{attribute 'linkalways'} 
{attribute 'no_explicit_call' := 'This FB is a CLASS and must be accessed using methods or properties'}
{attribute 'enable_dynamic_creation'}
FUNCTION_BLOCK _ETcVnDrawMatchesFlags EXTENDS EnumDatatypeBase
VAR
	localData : ETcVnDrawMatchesFlags;
	activeData : REFERENCE TO ETcVnDrawMatchesFlags;
	enumBaseDatatype : _DINT(localData);
END_VAR

METHOD PRIVATE AddLocalEnumeration
VAR_INPUT
	Enumeration : T_MAXSTRING;
	Value : ETcVnDrawMatchesFlags;
END_VAR
AddEnumeration(Enumeration, Value);
END_METHOD

PROPERTY PUBLIC Address : PVOID
GET
Address := ADR(activeData);
END_GET
END_PROPERTY

METHOD PUBLIC ClearReference
VAR_INPUT
END_VAR
activeData REF= localData;
SetBaseDatatypeReference();
END_METHOD

METHOD PUBLIC Clone : I_Datatype
VAR
    pClone : POINTER TO _ETcVnDrawMatchesFlags;
END_VAR
pClone := __NEW(_ETcVnDrawMatchesFlags(InitialValue := Value));
Clone := pClone^;
END_METHOD

METHOD FB_init : BOOL
VAR_INPUT
	bInitRetains : BOOL; // if TRUE, the retain variables are initialized (warm start / cold start)
	bInCopyCode : BOOL;  // if TRUE, the instance afterwards gets moved into the copy code (online change)
	InitialValue : ETcVnDrawMatchesFlags;
END_VAR
localData := InitialValue;
AddBaseDatatype(enumBaseDatatype);
ClearReference();

AddLocalEnumeration('TCVN_DMF_DEFAULT', ETcVnDrawMatchesFlags.TCVN_DMF_DEFAULT);
AddLocalEnumeration('TCVN_DMF_OVERDRAW', ETcVnDrawMatchesFlags.TCVN_DMF_OVERDRAW);
AddLocalEnumeration('TCVN_DMF_SKIPSINGLE', ETcVnDrawMatchesFlags.TCVN_DMF_SKIPSINGLE);
AddLocalEnumeration('TCVN_DMF_OVERDRAW_SKIPSINGLE', ETcVnDrawMatchesFlags.TCVN_DMF_OVERDRAW_SKIPSINGLE);
AddLocalEnumeration('TCVN_DMF_RICHKEYPOINT', ETcVnDrawMatchesFlags.TCVN_DMF_RICHKEYPOINT);
AddLocalEnumeration('TCVN_DMF_OVERDRAW_RICHKEYPOINT', ETcVnDrawMatchesFlags.TCVN_DMF_OVERDRAW_RICHKEYPOINT);
AddLocalEnumeration('TCVN_DMF_SKIPSINGLE_RICHKEYPOINT', ETcVnDrawMatchesFlags.TCVN_DMF_SKIPSINGLE_RICHKEYPOINT);
AddLocalEnumeration('TCVN_DMF_OVERDRAW_SKIPSINGLE_RICHKEYPOINT', ETcVnDrawMatchesFlags.TCVN_DMF_OVERDRAW_SKIPSINGLE_RICHKEYPOINT);
END_METHOD

PROPERTY PUBLIC Identifier : T_MAXSTRING
GET
Identifier := 'ETcVnDrawMatchesFlags';
END_GET
END_PROPERTY

METHOD IsEnumeratorValueEqual : BOOL
VAR_INPUT
	Enumerator : I_KeyValueForwardEnumerator;
END_VAR
VAR
	storedValue : ETcVnDrawMatchesFlags;
END_VAR
IF NOT Enumerator.TryGet(storedValue) THEN
	RETURN;
END_IF

IsEnumeratorValueEqual := storedValue = activeData;
END_METHOD

METHOD PUBLIC MakeReferenceTo
VAR_INPUT
	ReferenceTarget : REFERENCE TO ETcVnDrawMatchesFlags;
END_VAR
activeData REF= ReferenceTarget;
SetBaseDatatypeReference();
END_METHOD

METHOD PROTECTED SetBaseDatatypeReference
VAR_INPUT
END_VAR
enumBaseDatatype.MakeReferenceTo(activeData);
END_METHOD

PROPERTY PUBLIC Size : UDINT
GET
Size := SIZEOF(activeData);
END_GET
END_PROPERTY

METHOD TryMakeReferenceTo : BOOL
VAR_INPUT
	Target : I_Datatype;
END_VAR
VAR
	targetAsEnum : I_EnumDatatype;
	pTargetData : POINTER TO ETcVnDrawMatchesFlags;
END_VAR
IF NOT Target.TryResolveAsEnumDatatype(targetAsEnum) THEN
	RETURN;
END_IF

IF targetAsEnum.Identifier <> Identifier THEN
	RETURN;
END_IF

pTargetData := Target.Address;
activeData REF= pTargetData^;
SetBaseDatatypeReference();
TryMakeReferenceTo := TRUE;
END_METHOD

PROPERTY PUBLIC Value : ETcVnDrawMatchesFlags
GET
Value := activeData;
END_GET
SET
activeData := Value;
END_SET
END_PROPERTY

END_FUNCTION_BLOCK

(* stored: Version 1.1.0.1, ProductVersion 3.1.4024.12
   POU _ETcVnDrawMatchesFlags: Id {73629d68-2f5d-49ff-94a7-7ca7cec57a35}, SpecialFunc None
   Folder Constructor: Id {32d96447-e7f0-4675-9007-17a537760d92}
   Folder Private: Id {c680bf47-7463-46d6-af3a-9c0dd3f34d5f}
   Folder Protected: Id {e50697a4-5c03-45b7-b8c5-4a3b3ac778d9}
   Method AddLocalEnumeration: Id {dac81ec1-1941-4add-a8f9-5c7365b133b3}
   Property Address: Id {4dfc363e-885b-49cb-b25b-7bd2f073c2cc}
   Get Get: Id {1cea9c2e-8d6d-41bb-a799-155f0282aa03}
   Method ClearReference: Id {96e0f9db-7e13-465a-b546-4f0bad318b15}
   Method Clone: Id {e7c9abc3-d371-413a-ba76-f13805b09828}
   Method FB_init: Id {d9a5d8bc-4c45-46ba-ac38-a69413dff1e3}
   Property Identifier: Id {1c4343af-72c8-4423-a84b-952720d7bff0}
   Get Get: Id {541cafd0-444a-46cb-83c1-91e9079423cc}
   Method IsEnumeratorValueEqual: Id {5adcd422-e392-4d02-96e5-c18fc03fe199}
   Method MakeReferenceTo: Id {e4d459cb-c96b-42db-9005-038b3a8999d1}
   Method SetBaseDatatypeReference: Id {f9e79972-8cac-4663-b80a-036a249a0aca}
   Property Size: Id {777f2de3-8117-4c15-bb27-dfaf70785e0f}
   Get Get: Id {20a00256-d0b9-485e-9394-a2417d1faeb0}
   Method TryMakeReferenceTo: Id {ba2c7bb3-4e8b-4894-ac56-32d49e7e2378}
   Property Value: Id {08d529be-fbf2-41e9-963b-d1c576cd0f13}
   Get Get: Id {bdb87810-5f42-4f97-a76b-834854d01944}
   Set Set: Id {bd46c93f-f510-48f6-b779-ad56306f24b7} *)
